// TIA Portal V17 export
// export: Created 2024-03-30T11:14:40.1860502Z, ExportSetting WithDefaults, DisplayName Totally Integrated Automation Portal, DisplayVersion V17, DisplayName TIA Portal Openness, DisplayVersion V17, DisplayName TIA Portal Version Control Interface, DisplayVersion V17, DisplayName STEP 7 Professional, DisplayVersion V17, DisplayName STEP 7 Safety, DisplayVersion V17, DisplayName WinCC Advanced, DisplayVersion V17
DATA_BLOCK "gtyp_VGR"   // DB2
TITLE = Global DB VGR
{ S7_Optimized_Access := 'TRUE' }
AUTHOR : A.Schaefer
VERSION : 0.0
// stored: AutoNumber true, DBAccessibleFromOPCUA true, DBAccessibleFromWebserver true, InstanceOfName typ_VGR, InstanceOfType UDT, IsOnlyStoredInLoadMemory false, IsWriteProtectedInAS false
"typ_VGR"
   // VAR RETAIN
   //    x_Start_Park_Position : Bool;
   //    x_Park_Position_Reached : Bool;
   //    x_NFC_Start_First : Bool;
   //    x_NFC_Start : Bool;
   //    x_NFC_Completed : Bool;
   //    x_HBW_Storage : Bool;
   //    x_HBW_Outsource : Bool;
   //    s_HBW_Outsource_Typ : String;
   //    x_HBW_Discards : Bool;
   //    x_HBW_PickedUp : Bool;
   //    x_MPO_Req_Discard : Bool;
   //    x_MPO_Discards : Bool;
   //    x_Ready_For_Outsource : Bool;
   //    x_State_Process : Bool;
   //    x_Workpiece_NiO : Bool;
   //    horizontal_Axis : "typ_Axis";
   //    vertical_Axis : "typ_Axis";
   //    rotate_Axis : "typ_Axis";
   //    Workpiece : "typ_Workpiece";
   //    Worpiece_Parameters { S7_SetPoint := 'True'} : "typ_Workpiece_Parameters";
   //    History { S7_SetPoint := 'True'} : Array[1..20] of "typ_History";
   //    di_Pos_DSI_horizontal : DInt := 20;
   //    di_Pos_DSI_Collect_vertical : DInt := 2950;
   //    di_Pos_DSI_Discard_vertical : DInt;
   //    di_Offset_Pos_DSI_NFC_vertical : DInt := 1200;
   //    di_Pos_DSI_rotate : DInt := 20;
   //    di_Pos_DSO_horizontal : DInt := 2070;
   //    di_Pos_DSO_Collect_vertical : DInt;
   //    di_Pos_DSO_Discard_vertical : DInt := 1480;
   //    di_Offset_Pos_DSO_vertical : DInt := 500;
   //    di_Pos_DSO_rotate : DInt := 930;
   //    di_Pos_Color_horizontal : DInt := 150;
   //    di_Pos_Color_vertical : DInt := 2450;
   //    di_Pos_Color_rotate : DInt := 380;
   //    di_Pos_NFC_horizontal : DInt := 900;
   //    di_Pos_NFC_vertical : DInt := 2450;
   //    di_Pos_NFC_rotate : DInt := 680;
   //    di_Pos_MPO_horizontal : DInt := 3400;
   //    di_Pos_MPO_vertical : DInt := 1800;
   //    di_Offset_Pos_MPO_vertical : DInt := 650;
   //    di_Pos_MPO_rotate : DInt := 3480;
   //    di_Pos_Free_MPO_Min_rotate : DInt := 2500;
   //    di_Pos_Free_MPO_Max_rotate : DInt := 4000;
   //    di_Pos_Free_MPO_horizontal : DInt := 2000;
   //    di_Pos_HBW_horizontal : DInt := 600;
   //    di_Offset_Pos_HBW_horizontal : DInt;
   //    di_Pos_HBW_Collect_vertical : DInt := 650;
   //    di_Pos_HBW_Discard_vertical : DInt := 200;
   //    di_Offset_Pos_HBW_vertical : DInt := 100;
   //    di_Pos_HBW_rotate : DInt := 5330;
   //    di_Pos_NiO_horizontal : DInt;
   //    di_Pos_NiO_vertical : DInt := 2700;
   //    di_Pos_NiO_rotate : DInt := 1100;
   //    di_Pos_SLD_Blue_horizontal : DInt := 2150;
   //    di_Pos_SLD_Blue_vertical : DInt := 3100;
   //    di_Pos_SLD_Blue_rotate : DInt := 1160;
   //    di_Pos_SLD_Red_horizontal : DInt := 1580;
   //    di_Pos_SLD_Red_vertical : DInt := 3100;
   //    di_Pos_SLD_Red_rotate : DInt := 1430;
   //    di_Pos_SLD_White_horizontal : DInt := 1370;
   //    di_Pos_SLD_White_vertical : DInt := 3100;
   //    di_Pos_SLD_White_rotate : DInt := 1730;
   //    di_Pos_Park_horizontal : DInt := 150;
   //    di_Pos_Park_vertical : DInt := 3000;
   //    di_Pos_Park_rotate : DInt := 1750;
   //    x_Ready_For_Order : Bool;
   // END_VAR
BEGIN
   horizontal_Axis.i_PWM := -1;   // -1 sets auto PWM calculation
   horizontal_Axis.Config.di_Pos_Soft_Switch := 20000;
   vertical_Axis.i_PWM := -1;   // -1 sets auto PWM calculation
   vertical_Axis.Config.di_Pos_Soft_Switch := 20000;
   rotate_Axis.i_PWM := -1;   // -1 sets auto PWM calculation
   rotate_Axis.Config.di_Pos_Soft_Switch := 20000;
END_DATA_BLOCK
